// TIA Portal V20 export
DATA_BLOCK "InstEmOverviewHomeCondition"   // DB355
// stored: InstanceOfName EmOverviewHomeCondition, InstanceOfType FB
"EmOverviewHomeCondition"
   // VAR
   //    statMaxPageCount : Array[0..13] of Int;
   //    statPulse { ExternalAccessible := 'False'; ExternalVisible := 'False'; ExternalWritable := 'False'} : Array[0..199] of Bool;
   //    statLampOff { ExternalAccessible := 'False'; ExternalVisible := 'False'; ExternalWritable := 'False'} : Array[0..13] of Bool;
   //    statLampControl { ExternalAccessible := 'False'; ExternalVisible := 'False'; ExternalWritable := 'False'} : Bool;
   // END_VAR
BEGIN
END_DATA_BLOCK
